// TIA Portal V20 export
// export: Created 2025-12-01T14:56:12.0758501Z, ExportSetting None, DisplayName Totally Integrated Automation Portal, DisplayVersion V20 Update 3, DisplayName TIA Portal Openness, DisplayVersion V20 Update 3, DisplayName TIA Portal Version Control Interface, DisplayVersion V20 Update 3, DisplayName STEP 7 Professional, DisplayVersion V20 Update 3, DisplayName STEP 7 Safety, DisplayVersion V20 Update 2, DisplayName WinCC Basic/Comfort/Advanced, DisplayVersion V20 Update 3, DisplayName WinCC Professional, DisplayVersion V20 Update 3, DisplayName WinCC Unified, DisplayVersion V20 Update 3
TYPE "MoviManualMaquina"
   STRUCT
      Byte0_bit0 : Bool;   // ...
      Byte0_bit1 : Bool;   // ...
      Byte0_bit2 : Bool;   // ...
      Byte0_bit3 : Bool;   // ...
      Byte0_bit4 : Bool;   // ...
      Byte0_bit5 : Bool;   // ...
      Byte0_bit6 : Bool;   // ...
      Byte0_bit7 : Bool;   // ...
      Byte1_bit0 : Bool;   // ...
      Byte1_bit1 : Bool;   // ...
      Byte1_bit2 : Bool;   // ...
      Byte1_bit3 : Bool;   // ...
      Byte1_bit4 : Bool;   // ...
      Byte1_bit5 : Bool;   // ...
      Byte1_bit6 : Bool;   // ...
      Byte1_bit7 : Bool;   // ...
      Byte2_bit0 : Bool;   // ...
      Byte2_bit1 : Bool;   // ...
      Byte2_bit2 : Bool;   // ...
      Byte2_bit3 : Bool;   // ...
      Byte2_bit4 : Bool;   // ...
      Byte2_bit5 : Bool;   // ...
      Byte2_bit6 : Bool;   // ...
      Byte2_bit7 : Bool;   // ...
      Byte3_bit0 : Bool;   // ...
      Byte3_bit1 : Bool;   // ...
      Byte3_bit2 : Bool;   // ...
      Byte3_bit3 : Bool;   // ...
      Byte3_bit4 : Bool;   // ...
      Byte3_bit5 : Bool;   // ...
      Byte3_bit6 : Bool;   // ...
      Byte3_bit7 : Bool;   // ...
      Byte4_bit0 : Bool;   // ...
      Byte4_bit1 : Bool;   // ...
      Byte4_bit2 : Bool;   // ...
      Byte4_bit3 : Bool;   // ...
      Byte4_bit4 : Bool;   // ...
      Byte4_bit5 : Bool;   // ...
      Byte4_bit6 : Bool;   // ...
      Byte4_bit7 : Bool;   // ...
      Byte5_bit0 : Bool;   // ...
      Byte5_bit1 : Bool;   // ...
      Byte5_bit2 : Bool;   // ...
      Byte5_bit3 : Bool;   // ...
      Byte5_bit4 : Bool;   // ...
      Byte5_bit5 : Bool;   // ...
      Byte5_bit6 : Bool;   // ...
      Byte5_bit7 : Bool;   // ...
      Byte6_bit0 : Bool;   // ...
      Byte6_bit1 : Bool;   // ...
      Byte6_bit2 : Bool;   // ...
      Byte6_bit3 : Bool;   // ...
      Byte6_bit4 : Bool;   // ...
      Byte6_bit5 : Bool;   // ...
      Byte6_bit6 : Bool;   // ...
      Byte6_bit7 : Bool;   // ...
      Byte7_bit0 : Bool;   // ...
      Byte7_bit1 : Bool;   // ...
      Byte7_bit2 : Bool;   // ...
      Byte7_bit3 : Bool;   // ...
      Byte7_bit4 : Bool;   // ...
      Byte7_bit5 : Bool;   // ...
      Byte7_bit6 : Bool;   // ...
      Byte7_bit7 : Bool;   // ...
   END_STRUCT;
END_TYPE
